    rq_wait_ft_sensor_steady(2000)
    zero_ftsensor()
    sleep(0.1)
    # end: URCap Program Node
    # begin: URCap Program Node
    #   Source: Robotiq_Copilot, 1.22.1.14215, Robotiq Inc.
    #   Type: Find Surface
    $ 107 "Find Surface"
    zero_ftsensor()
    sleep(0.1)
    surface_found = rq_linear_search_urcap("Z+", 10.000, 0.005000, 0.100000, 1)
    storevar.setvariablepose("rq_findSurface_4f6a7ece-8f5f-4b59-9bc6-3e6f950945fc_exitPosition", get_actual_tcp_pose())
    $ 108 "'Add Stop conditions from the Find Surface node'" "noBreak"
    # 'Add Stop conditions from the Find Surface node'
    # end: URCap Program Node
    # begin: URCap Program Node
    #   Source: Robotiq_Copilot, 1.22.1.14215, Robotiq Inc.
    #   Type: Finishing Tool Control
    $ 109 "Start tool"
    set_standard_digital_out(0, True)
    # end: URCap Program Node
    $ 110 "Wait: 0.5"
    sleep(0.5)
    $ 111 "Force"
    sleep(0.02)
    zero_ftsensor()
    force_mode(tool_pose(), [0, 0, 1, 0, 0, 0], [0.0, 0.0, 5.0, 0.0, 0.0, 0.0], 2, [0.1, 0.1, 0.15, 0.3490658503988659, 0.3490658503988659, 0.3490658503988659])
    $ 112 "Waypoint_7" "noBreak"
    set_tcp(p[0.00318,0.11464,0.09820000000000001,-0.7853981633974483,0.0,0.0])
    movel(pose_trans(CubeFront, pose_trans(p[.002249871974, -.169402369556, .608081756259, .020435046430, 2.223511403835, 2.209446612627], Waypoint_7_p)), a=1.2, v=0.05)
    end_force_mode()
    stopl(5.0)
    # begin: URCap Program Node
    #   Source: Robotiq_Copilot, 1.22.1.14215, Robotiq Inc.
    #   Type: Finishing Tool Control
    $ 113 "Stop tool"
    set_standard_digital_out(0, False)
    # end: URCap Program Node
    $ 114 "Direction: CubeFront Z+"
    global move_thread_flag_114=0
    thread move_thread_114():
      enter_critical
      move_thread_flag_114 = 1
      local towardsPos=calculate_point_to_move_towards(p[-0.576714336693231,-0.2879231589673634,0.3016984353694383,1.2136593617103633,1.1943437168676707,1.19394259258799], [0.0,0.0,1.0], 0.05)
      movel(towardsPos, a=1.2, v=0.25)
      move_thread_flag_114 = 2
      exit_critical
    end
    move_thread_flag_114 = 0
    move_thread_han_114 = run move_thread_114()
    while (True):
      sleep(1.0E-10)
      if (move_thread_flag_114 > 1):
        join move_thread_han_114
        $ 115 "Until (distance)"
        break
      end
      sync()
    end
    $ 118 "Clear" "breakAfter"
    movej(Clear_q, a=1.3962634015954636, v=1.0471975511965976)
  end
  def SprayFront():
    $ 119 "SprayFront" "noBreak"
    $ 120 "SprayFront"
    $ 121 "MoveJ"
    $ 122 "SprayClear" "breakAfter"
    set_tcp(p[0.020839023181949995,-0.027139950822234082,0.10599373590389219,0.12258870209179472,1.1769383890382668,2.869747076630172])
    movej(get_inverse_kin(pose_trans(SprayPlane, pose_trans(p[.108036142494, -.305202473770, .810091201248, -1.216647948939, 1.210557871618, 1.204123812639], SprayClear_p)), qnear=SprayClear_q), a=1.3962634015954636, v=1.0471975511965976)
    $ 123 "MoveJ"
    $ 124 "Waypoint_10" "breakAfter"
    set_tcp(p[0.020839023181949995,-0.027139950822234082,0.10599373590389219,0.12258870209179472,1.1769383890382668,2.869747076630172])
    movej(get_inverse_kin(pose_trans(SprayPlane, pose_trans(p[.380158499114, -.183027591855, .571104219868, -1.574901506950, .032921162495, .010611987369], Waypoint_10_p)), qnear=Waypoint_10_q), a=1.3962634015954636, v=1.0471975511965976)
    $ 125 "Set DO[4]=On"
    set_standard_digital_out(4, True)
    $ 126 "MoveL"
    $ 127 "Waypoint_12" "breakAfter"
    movel(pose_trans(SprayPlane, pose_trans(p[.380158499114, -.183027591855, .571104219868, -1.574901506950, .032921162495, .010611987369], Waypoint_12_p)), a=1.2, v=0.1)
    $ 128 "Set DO[4]=Off"
    set_standard_digital_out(4, False)
    $ 129 "Direction: Tool Z-"
    global move_thread_flag_129=0
    thread move_thread_129():
      enter_critical
      move_thread_flag_129 = 1
      local towardsPos=calculate_point_to_move_towards(get_forward_kin(), [0.0,0.0,-1.0], 0.1)
      movel(towardsPos, a=1.2, v=0.2)
      move_thread_flag_129 = 2
      exit_critical
    end
    move_thread_flag_129 = 0
    move_thread_han_129 = run move_thread_129()
    while (True):
      sleep(1.0E-10)
      if (move_thread_flag_129 > 1):
        join move_thread_han_129
        $ 130 "Until (distance)"
        break
      end
      sync()
    end
    $ 131 "MoveJ"
    $ 132 "Waypoint_21" "breakAfter"
    set_tcp(p[0.020839023181949995,-0.027139950822234082,0.10599373590389219,0.12258870209179472,1.1769383890382668,2.869747076630172])
    movej(get_inverse_kin(pose_trans(SprayPlane, pose_trans(p[.380158499114, -.183027591855, .571104219868, -1.574901506950, .032921162495, .010611987369], Waypoint_21_p)), qnear=Waypoint_21_q), a=1.3962634015954636, v=1.0471975511965976)
    $ 133 "Set DO[4]=On"
    set_standard_digital_out(4, True)
    $ 134 "MoveL"
    $ 135 "Waypoint_22" "breakAfter"
    set_tcp(p[0.020839023181949995,-0.027139950822234082,0.10599373590389219,0.12258870209179472,1.1769383890382668,2.869747076630172])
    movel(pose_trans(SprayPlane, pose_trans(p[.380158499114, -.183027591855, .571104219868, -1.574901506950, .032921162495, .010611987369], Waypoint_22_p)), a=1.2, v=0.1)
    $ 136 "Set DO[4]=Off"
    set_standard_digital_out(4, False)
    $ 137 "Direction: Tool Z-"
    global move_thread_flag_137=0
    thread move_thread_137():
      enter_critical
      move_thread_flag_137 = 1
      local towardsPos=calculate_point_to_move_towards(get_forward_kin(), [0.0,0.0,-1.0], 0.1)
      movel(towardsPos, a=1.2, v=0.2)
      move_thread_flag_137 = 2
      exit_critical
    end
    move_thread_flag_137 = 0
    move_thread_han_137 = run move_thread_137()
    while (True):
      sleep(1.0E-10)
      if (move_thread_flag_137 > 1):
        join move_thread_han_137
        $ 138 "Until (distance)"
        break
      end
      sync()
    end
    $ 139 "MoveJ"
    $ 140 "Waypoint_23" "breakAfter"
    set_tcp(p[0.020839023181949995,-0.027139950822234082,0.10599373590389219,0.12258870209179472,1.1769383890382668,2.869747076630172])
    movej(get_inverse_kin(pose_trans(SprayPlane, pose_trans(p[.200894234219, -.299948761986, .678711619414, -1.215428189557, 1.212361481441, 1.193485326269], Waypoint_23_p)), qnear=Waypoint_23_q), a=1.3962634015954636, v=1.0471975511965976)
    $ 141 "Set DO[4]=On"
    set_standard_digital_out(4, True)
    $ 142 "MoveL"
    $ 143 "Waypoint_24" "breakAfter"
    set_tcp(p[0.020839023181949995,-0.027139950822234082,0.10599373590389219,0.12258870209179472,1.1769383890382668,2.869747076630172])
    movel(pose_trans(SprayPlane, pose_trans(p[.200894234219, -.299948761986, .678711619414, -1.215428189557, 1.212361481441, 1.193485326269], Waypoint_24_p)), a=1.2, v=0.1)
    $ 144 "Set DO[4]=Off"
    set_standard_digital_out(4, False)
    $ 145 "Direction: Tool Z-"
    global move_thread_flag_145=0
    thread move_thread_145():
      enter_critical
      move_thread_flag_145 = 1
      local towardsPos=calculate_point_to_move_towards(get_forward_kin(), [0.0,0.0,-1.0], 0.1)
      movel(towardsPos, a=1.2, v=0.2)
      move_thread_flag_145 = 2
      exit_critical
    end
    move_thread_flag_145 = 0
    move_thread_han_145 = run move_thread_145()
    while (True):
      sleep(1.0E-10)
      if (move_thread_flag_145 > 1):
        join move_thread_han_145
        $ 146 "Until (distance)"
        break
      end
      sync()
    end
    $ 147 "Direction: Base Z+"
    global move_thread_flag_147=0
    thread move_thread_147():
      enter_critical
      move_thread_flag_147 = 1
      local towardsPos=calculate_point_to_move_towards(p[0.0,0.0,0.0,0.0,0.0,0.0], [0.0,0.0,1.0], 0.1)
      movel(towardsPos, a=1.2, v=0.1)
      move_thread_flag_147 = 2
      exit_critical
    end
    move_thread_flag_147 = 0
    move_thread_han_147 = run move_thread_147()
    while (True):
      sleep(1.0E-10)
      if (move_thread_flag_147 > 1):
        join move_thread_han_147
        $ 148 "Until (distance)"
        break
      end
      sync()
    end
    $ 149 "MoveJ"
    $ 150 "Waypoint_38" "breakAfter"
    set_tcp(p[0.020839023181949995,-0.027139950822234082,0.10599373590389219,0.12258870209179472,1.1769383890382668,2.869747076630172])
    movej(get_inverse_kin(pose_trans(SprayPlane, pose_trans(p[.152076837040, -.186455621862, .570552501782, -1.567181840228, .028822735400, .008142754325], Waypoint_38_p)), qnear=Waypoint_38_q), a=1.3962634015954636, v=1.0471975511965976)
    $ 151 "Set DO[4]=On"
    set_standard_digital_out(4, True)
    $ 152 "MoveL"
    $ 153 "Waypoint_25" "breakAfter"
    set_tcp(p[0.020839023181949995,-0.027139950822234082,0.10599373590389219,0.12258870209179472,1.1769383890382668,2.869747076630172])
    movel(pose_trans(SprayPlane, pose_trans(p[.380158499114, -.183027591855, .571104219868, -1.574901506950, .032921162495, .010611987369], Waypoint_25_p)), a=1.2, v=0.1)
    $ 154 "Set DO[4]=Off"
    set_standard_digital_out(4, False)
    $ 155 "Direction: Tool Z-"
    global move_thread_flag_155=0
    thread move_thread_155():
      enter_critical
      move_thread_flag_155 = 1
      local towardsPos=calculate_point_to_move_towards(get_forward_kin(), [0.0,0.0,-1.0], 0.1)
      movel(towardsPos, a=1.2, v=0.2)
      move_thread_flag_155 = 2
      exit_critical
    end
    move_thread_flag_155 = 0
    move_thread_han_155 = run move_thread_155()
    while (True):
      sleep(1.0E-10)
      if (move_thread_flag_155 > 1):
        join move_thread_han_155
        $ 156 "Until (distance)"
        break
      end
      sync()
    end
    $ 157 "MoveJ"
    $ 158 "SprayClear" "breakAfter"
    set_tcp(p[0.020839023181949995,-0.027139950822234082,0.10599373590389219,0.12258870209179472,1.1769383890382668,2.869747076630172])
    movej(get_inverse_kin(pose_trans(SprayPlane, pose_trans(p[.108036142494, -.305202473770, .810091201248, -1.216647948939, 1.210557871618, 1.204123812639], SprayClear_p)), qnear=SprayClear_q), a=1.3962634015954636, v=1.0471975511965976)
  end
  def SprayRebate():
    $ 159 "SprayRebate" "noBreak"
    $ 160 "SprayRebate"
    $ 161 "MoveJ"
    $ 162 "SprayClear" "breakAfter"
    set_tcp(p[0.020839023181949995,-0.027139950822234082,0.10599373590389219,0.12258870209179472,1.1769383890382668,2.869747076630172])
    movej(get_inverse_kin(pose_trans(SprayPlane, pose_trans(p[.108036142494, -.305202473770, .810091201248, -1.216647948939, 1.210557871618, 1.204123812639], SprayClear_p)), qnear=SprayClear_q), a=1.3962634015954636, v=1.0471975511965976)
    $ 163 "MoveJ"
    $ 164 "Waypoint_28" "breakAfter"
    set_tcp(p[0.020839023181949995,-0.027139950822234082,0.10599373590389219,0.12258870209179472,1.1769383890382668,2.869747076630172])
    movej(get_inverse_kin(pose_trans(SprayPlane, pose_trans(p[-.002001169423, -.178123008725, .618090231485, -1.568699287997, .013964727372, .007428573496], Waypoint_28_p)), qnear=Waypoint_28_q), a=1.3962634015954636, v=1.0471975511965976)
    $ 165 "Set DO[4]=On"
    set_standard_digital_out(4, True)
    $ 166 "MoveL"
    $ 167 "Waypoint_27" "breakAfter"
    set_tcp(p[0.020839023181949995,-0.027139950822234082,0.10599373590389219,0.12258870209179472,1.1769383890382668,2.869747076630172])
    movel(pose_trans(SprayPlane, pose_trans(p[-.002001169423, -.178123008725, .618090231485, -1.568699287997, .013964727372, .007428573496], Waypoint_27_p)), a=1.2, v=0.1)
    $ 168 "Set DO[4]=Off"
    set_standard_digital_out(4, False)
    $ 169 "Direction: CubeFront Z-"
    global move_thread_flag_169=0
    thread move_thread_169():
      enter_critical
      move_thread_flag_169 = 1
      local towardsPos=calculate_point_to_move_towards(p[-0.576714336693231,-0.2879231589673634,0.3016984353694383,1.2136593617103633,1.1943437168676707,1.19394259258799], [0.0,0.0,-1.0], 0.2)
      movel(towardsPos, a=1.2, v=0.2)
      move_thread_flag_169 = 2
      exit_critical
    end
    move_thread_flag_169 = 0
    move_thread_han_169 = run move_thread_169()
    while (True):
      sleep(1.0E-10)
      if (move_thread_flag_169 > 1):
        join move_thread_han_169
        $ 170 "Until (distance)"
        break
      end
      sync()
    end
    $ 171 "MoveJ"
    $ 172 "Waypoint_29" "breakAfter"
    set_tcp(p[0.020839023181949995,-0.027139950822234082,0.10599373590389219,0.12258870209179472,1.1769383890382668,2.869747076630172])
    movej(get_inverse_kin(pose_trans(SprayPlane, pose_trans(p[-.002001169423, -.178123008725, .618090231485, -1.568699287997, .013964727372, .007428573496], Waypoint_29_p)), qnear=Waypoint_29_q), a=1.3962634015954636, v=1.0471975511965976)
    $ 173 "Set DO[4]=On"
    set_standard_digital_out(4, True)
    $ 174 "MoveL"
    $ 175 "Waypoint_30" "breakAfter"
    set_tcp(p[0.020839023181949995,-0.027139950822234082,0.10599373590389219,0.12258870209179472,1.1769383890382668,2.869747076630172])
    movel(pose_trans(SprayPlane, pose_trans(p[-.002001169423, -.178123008725, .618090231485, -1.568699287997, .013964727372, .007428573496], Waypoint_30_p)), a=1.2, v=0.1)
    $ 176 "Set DO[4]=Off"
    set_standard_digital_out(4, False)
    $ 177 "Direction: CubeFront Z-"
    global move_thread_flag_177=0
    thread move_thread_177():
      enter_critical
      move_thread_flag_177 = 1
      local towardsPos=calculate_point_to_move_towards(p[-0.576714336693231,-0.2879231589673634,0.3016984353694383,1.2136593617103633,1.1943437168676707,1.19394259258799], [0.0,0.0,-1.0], 0.2)
      movel(towardsPos, a=1.2, v=0.2)
      move_thread_flag_177 = 2
      exit_critical
    end
    move_thread_flag_177 = 0
    move_thread_han_177 = run move_thread_177()
    while (True):
      sleep(1.0E-10)
      if (move_thread_flag_177 > 1):
        join move_thread_han_177
        $ 178 "Until (distance)"
        break
      end
      sync()
    end
    $ 179 "MoveJ"
    $ 180 "SprayClear" "breakAfter"
    set_tcp(p[0.020839023181949995,-0.027139950822234082,0.10599373590389219,0.12258870209179472,1.1769383890382668,2.869747076630172])
    movej(get_inverse_kin(pose_trans(SprayPlane, pose_trans(p[.108036142494, -.305202473770, .810091201248, -1.216647948939, 1.210557871618, 1.204123812639], SprayClear_p)), qnear=SprayClear_q), a=1.3962634015954636, v=1.0471975511965976)
    $ 181 "MoveL"
    $ 182 "Direction: CubeFront Z-"
    global move_thread_flag_182=0
    thread move_thread_182():
      enter_critical
      move_thread_flag_182 = 1
      local towardsPos=calculate_point_to_move_towards(p[-0.576714336693231,-0.2879231589673634,0.3016984353694383,1.2136593617103633,1.1943437168676707,1.19394259258799], [0.0,0.0,-1.0], 0.1)
      movel(towardsPos, a=1.2, v=0.2)
      move_thread_flag_182 = 2
      exit_critical
    end
    move_thread_flag_182 = 0
    move_thread_han_182 = run move_thread_182()
    while (True):
      sleep(1.0E-10)
      if (move_thread_flag_182 > 1):
        join move_thread_han_182
        $ 183 "Until (distance)"
        break
      end
      sync()
    end
    $ 184 "MoveJ"
    $ 185 "Waypoint_32" "breakAfter"
    set_tcp(p[0.020839023181949995,-0.027139950822234082,0.10599373590389219,0.12258870209179472,1.1769383890382668,2.869747076630172])
    movej(get_inverse_kin(pose_trans(SprayPlane, pose_trans(p[-.002001169423, -.178123008725, .618090231485, -1.568699287997, .013964727372, .007428573496], Waypoint_32_p)), qnear=Waypoint_32_q), a=1.3962634015954636, v=1.0471975511965976)
    $ 186 "Set DO[4]=On"
    set_standard_digital_out(4, True)
    $ 187 "MoveL"
    $ 188 "Waypoint_33" "breakAfter"
    set_tcp(p[0.020839023181949995,-0.027139950822234082,0.10599373590389219,0.12258870209179472,1.1769383890382668,2.869747076630172])
    movel(pose_trans(SprayPlane, pose_trans(p[-.002001169423, -.178123008725, .618090231485, -1.568699287997, .013964727372, .007428573496], Waypoint_33_p)), a=1.2, v=0.1)
    $ 189 "Set DO[4]=Off"
    set_standard_digital_out(4, False)
    $ 190 "Direction: CubeFront Z-"
    global move_thread_flag_190=0
    thread move_thread_190():
      enter_critical
      move_thread_flag_190 = 1
      local towardsPos=calculate_point_to_move_towards(p[-0.576714336693231,-0.2879231589673634,0.3016984353694383,1.2136593617103633,1.1943437168676707,1.19394259258799], [0.0,0.0,-1.0], 0.2)
      movel(towardsPos, a=1.2, v=0.2)
      move_thread_flag_190 = 2
      exit_critical
    end
    move_thread_flag_190 = 0
    move_thread_han_190 = run move_thread_190()
    while (True):
      sleep(1.0E-10)
      if (move_thread_flag_190 > 1):
        join move_thread_han_190
        $ 191 "Until (distance)"
        break
      end
      sync()
    end
    $ 192 "MoveJ"
    $ 193 "SprayClear" "breakAfter"
    set_tcp(p[0.020839023181949995,-0.027139950822234082,0.10599373590389219,0.12258870209179472,1.1769383890382668,2.869747076630172])
    movej(get_inverse_kin(pose_trans(SprayPlane, pose_trans(p[.108036142494, -.305202473770, .810091201248, -1.216647948939, 1.210557871618, 1.204123812639], SprayClear_p)), qnear=SprayClear_q), a=1.3962634015954636, v=1.0471975511965976)
  end
  def SandFront():
    $ 194 "SandFront" "noBreak"
    $ 195 "sandFront"
    $ 196 "MoveJ"
    $ 197 "Clear" "breakAfter"
    movej(Clear_q, a=1.3962634015954636, v=1.0471975511965976)
    $ 199 "MoveL"
    $ 200 "Waypoint_1" "breakAfter"
    set_tcp(p[0.00318,0.11464,0.09820000000000001,-0.7853981633974483,0.0,0.0])
    movel(pose_trans(Work, pose_trans(p[-.005597006121, -.192408094989, .653246871754, -1.571622694982, -.002967386491, .002471774867], Waypoint_1_p)), a=1.2, v=0.25)
    # begin: URCap Program Node
    #   Source: Robotiq_Copilot, 1.22.1.14215, Robotiq Inc.
    #   Type: Zero FT Sensor
    $ 201 "Zero FT Sensor"

    rq_wait_ft_sensor_steady(2000)
    zero_ftsensor()
    sleep(0.1)
    # end: URCap Program Node
    # begin: URCap Program Node
    #   Source: Robotiq_Copilot, 1.22.1.14215, Robotiq Inc.
    #   Type: Find Surface
    $ 202 "Find Surface"
    surface_found = rq_linear_search_urcap("Z+", 10.000, 0.005000, 0.100000, 1)
    storevar.setvariablepose("rq_findSurface_23f4c747-ad10-472d-8dd5-9c0057261c1a_exitPosition", get_actual_tcp_pose())
    $ 203 "'Add Stop conditions from the Find Surface node'" "noBreak"
    # 'Add Stop conditions from the Find Surface node'
    # end: URCap Program Node
    # begin: URCap Program Node
    #   Source: Robotiq_Copilot, 1.22.1.14215, Robotiq Inc.
    #   Type: Finishing Tool Control
    $ 204 "Start tool"
    set_standard_digital_out(0, True)
    # end: URCap Program Node
    $ 205 "Wait: 0.5"
    sleep(0.5)
    $ 206 "MoveL"
    $ 207 "Force"
    sleep(0.02)
    zero_ftsensor()
    force_mode(tool_pose(), [0, 0, 1, 0, 0, 0], [0.0, 0.0, 7.0, 0.0, 0.0, 0.0], 2, [0.1, 0.1, 0.15, 0.3490658503988659, 0.3490658503988659, 0.3490658503988659])
    $ 208 "Waypoint_34" "noBreak"
    set_tcp(p[0.00318,0.11464,0.09820000000000001,-0.7853981633974483,0.0,0.0])
    movel(pose_trans(Work, pose_trans(p[.002249871974, -.169402369556, .608081756259, .020435046430, 2.223511403835, 2.209446612627], Waypoint_34_p)), a=1.2, v=0.06)
    $ 209 "Waypoint_37" "noBreak"
    set_tcp(p[0.00318,0.11464,0.09820000000000001,-0.7853981633974483,0.0,0.0])
    movel(pose_trans(Work, pose_trans(p[.002249871974, -.169402369556, .608081756259, .020435046430, 2.223511403835, 2.209446612627], Waypoint_37_p)), a=1.2, v=0.06)
    $ 210 "Waypoint_36" "noBreak"
    set_tcp(p[0.00318,0.11464,0.09820000000000001,-0.7853981633974483,0.0,0.0])
    movel(pose_trans(Work, pose_trans(p[.002249871974, -.169402369556, .608081756259, .020435046430, 2.223511403835, 2.209446612627], Waypoint_36_p)), a=1.2, v=0.06)
    $ 211 "Waypoint_1" "noBreak"
    set_tcp(p[0.00318,0.11464,0.09820000000000001,-0.7853981633974483,0.0,0.0])
    movel(pose_trans(Work, pose_trans(p[-.005597006121, -.192408094989, .653246871754, -1.571622694982, -.002967386491, .002471774867], Waypoint_1_p)), a=1.2, v=0.06)
    # begin: URCap Program Node
    #   Source: Robotiq_Copilot, 1.22.1.14215, Robotiq Inc.
    #   Type: Finishing Tool Control
    $ 212 "Stop tool" "noBreak"
    set_standard_digital_out(0, False)
    # end: URCap Program Node
    end_force_mode()
    stopl(5.0)
    $ 213 "Direction: Tool Z-"
    global move_thread_flag_213=0
    thread move_thread_213():
      enter_critical
      move_thread_flag_213 = 1
      local towardsPos=calculate_point_to_move_towards(get_forward_kin(), [0.0,0.0,-1.0], 0.025)
      movel(towardsPos, a=1.2, v=0.06)
      move_thread_flag_213 = 2
      exit_critical
    end
    move_thread_flag_213 = 0
    move_thread_han_213 = run move_thread_213()
    while (True):
      sleep(1.0E-10)
      if (move_thread_flag_213 > 1):
        join move_thread_han_213
        $ 214 "Until (distance)"
        break
      end
      sync()
    end
    $ 215 "MoveJ"
    $ 216 "Clear" "breakAfter"
    movej(Clear_q, a=1.3962634015954636, v=1.0471975511965976)
  end
  def StartSpray():
    $ 218 "StartSpray" "noBreak"
    $ 219 "Set DO[1]=On"
    set_standard_digital_out(1, True)
    $ 220 "Wait: 0.3"
    sleep(0.3)
  end
  def stopSpray():
    $ 221 "stopSpray" "noBreak"
    $ 222 "Set DO[1]=Off"
    set_standard_digital_out(1, False)
    $ 223 "Wait: 0.3"
    sleep(0.3)
  end
  thread EventThread():
    while (True):
      if (get_standard_digital_in(0) !=   True  ):
        $ 60 "Set DO[0]=Off"
        set_standard_digital_out(0, False)
        $ 61 "Set DO[1]=Off"
        set_standard_digital_out(1, False)
        $ 62 "Halt"
        halt
      elif (get_standard_digital_in(1) ==   True  ):
        $ 64 "readyFrontSand≔ True "
        global readyFrontSand=  True
        $ 65 "Set DO[5]=On"
        set_standard_digital_out(5, True)
      elif (get_standard_digital_in(2) ==   True  ):
        $ 67 "readyBackSand≔ True "
        global readyBackSand=  True
        $ 68 "Set DO[5]=On"
        set_standard_digital_out(5, True)
      elif (get_standard_digital_in(3) ==   True  ):
        $ 70 "readySpray≔ True "
        global readySpray=  True
      end
      sync()
    end
  end
  eventThread = run EventThread()
  while (True):
    $ 2 "Robot Program"
    $ 3 "Main"
    $ 4 "If readyFrontSand≟ True "
    global thread_flag_4=0
    thread Thread_if_4():
      $ 5 "MoveJ"
      $ 6 "Clear" "breakAfter"
      movej(Clear_q, a=1.3962634015954636, v=1.0471975511965976)
      # begin: URCap Program Node
      #   Source: Robotiq_Copilot, 1.22.1.14215, Robotiq Inc.
      #   Type: Zero FT Sensor
      $ 7 "Zero FT Sensor"

      rq_wait_ft_sensor_steady(2000)
      zero_ftsensor()
      sleep(0.1)
      # end: URCap Program Node
      $ 8 "Work≔CubeFront"
      global Work=CubeFront
      $ 9 "Call SandFront"
      SandFront()
      $ 10 "Call SandRebate"
      SandRebate()
      $ 11 "readyFrontSand≔ False "
      global readyFrontSand=  False
      $ 12 "Set DO[5]=Off"
      set_standard_digital_out(5, False)
      thread_flag_4 = 1
    end
    if (readyFrontSand ==   True  ):
      global thread_handler_4=run Thread_if_4()
      while (thread_flag_4 == 0):
        if not(readyFrontSand ==   True  ):
          kill thread_handler_4
          thread_flag_4 = 2
        else:
          sync()
        end
      end
    else:
      thread_flag_4 = 2
    end
    $ 13 "If readyBackSand≟ True "
    global thread_flag_13=0
    thread Thread_if_13():
      $ 14 "Work≔CubeFront"
      global Work=CubeFront
      $ 15 "Call SandFront"
      SandFront()
      $ 16 "readyBackSand≔ False "
      global readyBackSand=  False
      $ 17 "Set DO[5]=Off"
      set_standard_digital_out(5, False)
      thread_flag_13 = 1
    end
    if (readyBackSand ==   True  ):
      global thread_handler_13=run Thread_if_13()
      while (thread_flag_13 == 0):
        if not(readyBackSand ==   True  ):
          kill thread_handler_13
          thread_flag_13 = 2
        else:
          sync()
        end
      end
    else:
      thread_flag_13 = 2
    end
    $ 18 "If readySpray≟ True "
    global thread_flag_18=0
    thread Thread_if_18():
      $ 19 "MoveJ"
      $ 20 "Waypoint_6" "breakAfter"
      movej(Waypoint_6_q, a=1.3962634015954636, v=1.0471975511965976)
      $ 21 "SprayClear" "breakAfter"
      movej(SprayClear_q, a=1.3962634015954636, v=1.0471975511965976)
      # begin: URCap Program Node
      #   Source: Robotiq_Copilot, 1.22.1.14215, Robotiq Inc.
      #   Type: Zero FT Sensor
      $ 22 "Zero FT Sensor"

      rq_wait_ft_sensor_steady(2000)
      zero_ftsensor()
      sleep(0.1)
      # end: URCap Program Node
      $ 23 "Call SprayFront"
      SprayFront()
      $ 24 "Call SprayRebate"
      SprayRebate()
      $ 25 "Waypoint_6" "breakAfter"
      movej(Waypoint_6_q, a=1.3962634015954636, v=1.0471975511965976)
      $ 26 "readySpray≔ False "
      global readySpray=  False
      thread_flag_18 = 1
    end
    if (readySpray ==   True  ):
      global thread_handler_18=run Thread_if_18()
      while (thread_flag_18 == 0):
        if not(readySpray ==   True  ):
          kill thread_handler_18
          thread_flag_18 = 2
        else:
          sync()
        end
      end
    else:
      thread_flag_18 = 2
    end
  end
end
